// Mitsubishi GX Works2 project: 0715지수표시   PLC: Q02/Q02H

PROGRAM MAIN
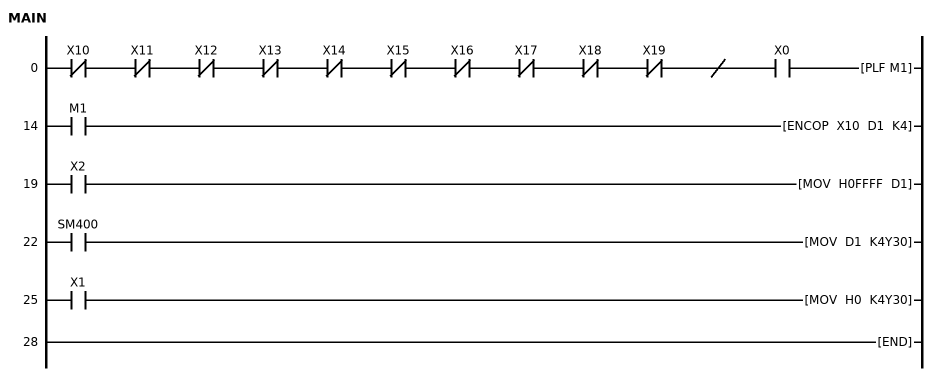
0     LDI     X10
      ANI     X11
      ANI     X12
      ANI     X13
      ANI     X14
      ANI     X15
      ANI     X16
      ANI     X17
      ANI     X18
      ANI     X19
      INV
      AND     X0
      PLF     M1
14    LD      M1
      ENCOP   X10 D1 K4
19    LD      X2
      MOV     H0FFFF D1
22    LD      SM400
      MOV     D1 K4Y30
25    LD      X1
      MOV     H0 K4Y30
28    END
END_PROGRAM
